{attribute 'qualified_only'}
{attribute 'strict'}
TYPE ST_BoxStatus :
(
	enum_member := 0
);
END_TYPE

(* stored: Version 1.1.0.1, ProductVersion 3.1.4024.13
   DUT ST_BoxStatus: Id {9a170bca-f7df-41a7-87ed-0da4027b5acc} *)
